Yaskawa INFORM job: long_pipe_cylinder_program.JBI

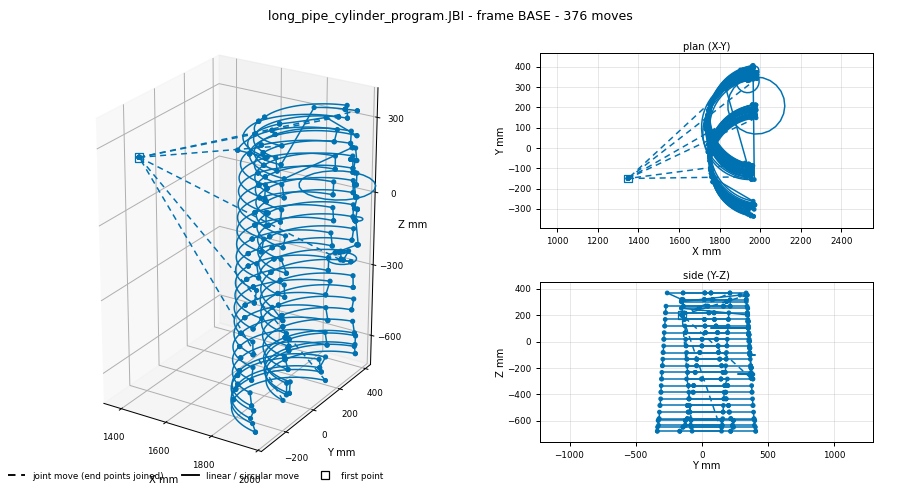
[picture p0: tool path of long_pipe_cylinder_program.JBI in frame BASE, 376 of 498 moves have a stored position in this frame; points joined in program order, loops and branches not executed]
/JOB
//NAME long_pipe_cylinder_program
//POS
///NPOS 488,0,488,1,0,4
///TOOL 0
///POSTYPE BASE
///RECTAN
///RCONF 0,0,0,0,0,0,0,0,0,0,0,0,0,0,0,0,0,0,0,0,0,0,0,0
C00000=1952.474,-141.608,367.212,-93.9778,-89.9999,5.0000
C00001=1952.474,-141.608,367.212,-93.9778,-89.9999,5.0000
C00002=1806.020,-80.138,367.212,-131.5952,-89.9999,5.0000
C00003=1753.400,68.522,367.212,-170.6555,-89.9999,5.0000
C00004=1753.400,68.522,367.212,-170.6555,-89.9999,5.0000
C00005=1753.400,68.522,367.212,-170.6555,-89.9999,5.0000
C00006=1795.925,238.470,367.212,142.2632,-89.9999,5.0000
C00007=1945.817,334.393,367.212,95.8859,-90.0000,5.0000
C00008=1947.913,335.229,317.245,95.3503,-90.0000,5.0000
C00009=1947.913,335.229,317.245,95.3503,-90.0000,5.0000
C00010=1748.482,181.577,317.245,160.6849,-90.0000,5.0000
C00011=1744.683,18.104,317.245,-159.0744,-89.9999,5.0000
C00012=1744.683,18.104,317.245,-159.0744,-89.9999,5.0000
C00013=1744.683,18.104,317.245,-159.0744,-89.9999,5.0000
C00014=1842.190,-106.459,317.245,-121.1710,-89.9999,5.0000
C00015=1928.137,-141.549,317.245,-99.5716,-90.0000,5.0000
C00016=1932.899,-139.870,267.245,-98.5458,-90.0000,5.0000
C00017=1932.899,-139.870,267.245,-98.5458,-90.0000,5.0000
C00018=1770.352,-30.060,267.245,-146.0425,-90.0000,5.0000
C00019=1741.797,163.121,267.245,165.4703,-89.9999,5.0000
C00020=1741.797,163.121,267.245,165.4703,-89.9999,5.0000
C00021=1741.797,163.121,267.245,165.4703,-89.9999,5.0000
C00022=1814.919,283.253,267.245,130.7984,-90.0000,5.0000
C00023=1962.193,340.769,267.245,91.7826,-90.0000,5.0000
C00024=1958.817,343.549,217.245,92.5686,-89.9999,5.0000
C00025=1958.817,343.549,217.245,92.5686,-89.9999,5.0000
C00026=1797.784,264.676,217.245,136.9283,-89.9999,5.0000
C00027=1734.064,92.078,217.245,-177.0797,-89.9999,5.0000
C00028=1734.064,92.078,217.245,-177.0797,-89.9999,5.0000
C00029=1734.064,92.078,217.245,-177.0797,-89.9999,5.0000
C00030=1799.958,-65.427,217.245,-135.0139,-90.0000,5.0000
C00031=1949.378,-134.142,217.245,-94.8421,-90.0000,5.0000
C00032=1957.810,-131.244,167.245,-92.8582,-90.0000,5.0000
C00033=1957.810,-131.244,167.245,-92.8582,-90.0000,5.0000
C00034=1801.335,-64.041,167.245,-135.0154,-89.9999,5.0000
C00035=1735.186,94.868,167.245,-177.7463,-90.0000,5.0000
C00036=1735.186,94.868,167.245,-177.7463,-90.0000,5.0000
C00037=1735.186,94.868,167.245,-177.7463,-90.0000,5.0000
C00038=1799.120,267.709,167.245,136.1700,-90.0000,5.0000
C00039=1966.952,347.413,167.245,90.6138,-90.0000,5.0000
C00040=1967.186,350.732,117.245,90.5513,-90.0000,5.0000
C00041=1967.186,350.732,117.245,90.5513,-90.0000,5.0000
C00042=1802.303,274.899,117.245,134.3981,-89.9999,5.0000
C00043=1734.310,106.876,117.245,179.3219,-89.9999,5.0000
C00044=1734.310,106.876,117.245,179.3219,-89.9999,5.0000
C00045=1734.310,106.876,117.245,179.3219,-89.9999,5.0000
C00046=1803.371,-61.994,117.245,-135.0176,-90.0000,5.0000
C00047=1945.844,-127.883,117.245,-95.8371,-90.0000,5.0000
C00048=1938.801,-124.320,67.245,-97.6695,-90.0000,5.0000
C00049=1938.801,-124.320,67.245,-97.6695,-90.0000,5.0000
C00050=1793.896,-48.619,67.245,-138.9983,-90.0000,5.0000
C00051=1735.617,118.587,67.245,176.4544,-89.9999,5.0000
C00052=1735.617,118.587,67.245,176.4544,-89.9999,5.0000
C00053=1735.617,118.587,67.245,176.4544,-89.9999,5.0000
C00054=1810.878,284.290,67.245,131.3668,-89.9999,5.0000
C00055=1968.204,353.422,67.245,90.3114,-90.0000,5.0000
C00056=1966.949,356.620,17.245,90.5922,-90.0000,5.0000
C00057=1966.949,356.620,17.245,90.5922,-90.0000,5.0000
C00058=1807.041,282.224,17.245,132.3756,-90.0000,5.0000
C00059=1736.566,110.516,17.245,178.4205,-89.9999,5.0000
C00060=1736.566,110.516,17.245,178.4205,-89.9999,5.0000
C00061=1736.566,110.516,17.245,178.4205,-89.9999,5.0000
C00062=1795.050,-47.099,17.245,-139.0948,-90.0000,5.0000
C00063=1959.444,-122.297,17.245,-92.5584,-90.0000,5.0000
C00064=1947.518,-118.948,-32.755,-95.6438,-90.0000,5.0000
C00065=1947.518,-118.948,-32.755,-95.6438,-90.0000,5.0000
C00066=1796.790,-44.821,-32.755,-139.2413,-89.9999,5.0000
C00067=1737.499,122.501,-32.755,175.4642,-90.0000,5.0000
C00068=1737.499,122.501,-32.755,175.4642,-90.0000,5.0000
C00069=1737.499,122.501,-32.755,175.4642,-90.0000,5.0000
C00070=1805.960,284.348,-32.755,132.2266,-89.9999,5.0000
C00071=1967.957,359.139,-32.755,90.3599,-89.9999,5.0000
C00072=1966.253,361.510,-82.755,90.7359,-90.0000,5.0000
C00073=1966.253,361.510,-82.755,90.7359,-90.0000,5.0000
C00074=1815.299,294.981,-82.755,128.9422,-89.9999,5.0000
C00075=1738.257,125.322,-82.755,174.7557,-90.0000,5.0000
C00076=1738.257,125.322,-82.755,174.7557,-90.0000,5.0000
C00077=1738.257,125.322,-82.755,174.7557,-90.0000,5.0000
C00078=1798.652,-42.311,-82.755,-139.4159,-90.0000,5.0000
C00079=1937.806,-115.431,-82.755,-98.2307,-90.0000,5.0000
C00080=1959.669,-113.835,-132.755,-92.5986,-90.0000,5.0000
C00081=1959.669,-113.835,-132.755,-92.5986,-90.0000,5.0000
C00082=1789.517,-29.714,-132.755,-143.3805,-89.9999,5.0000
C00083=1738.347,134.581,-132.755,172.4879,-89.9999,5.0000
C00084=1738.347,134.581,-132.755,172.4879,-89.9999,5.0000
C00085=1738.347,134.581,-132.755,172.4879,-89.9999,5.0000
C00086=1815.608,296.473,-132.755,128.6681,-89.9999,5.0000
C00087=1967.823,365.446,-132.755,90.3807,-90.0000,5.0000
C00088=1960.178,368.374,-182.755,92.0329,-90.0000,5.0000
C00089=1960.178,368.374,-182.755,92.0329,-90.0000,5.0000
C00090=1822.990,305.437,-182.755,126.0528,-90.0000,5.0000
C00091=1740.856,149.131,-182.755,168.8590,-90.0000,5.0000
C00092=1740.856,149.131,-182.755,168.8590,-90.0000,5.0000
C00093=1740.856,149.131,-182.755,168.8590,-90.0000,5.0000
C00094=1790.084,-24.585,-182.755,-144.3607,-90.0000,5.0000
C00095=1949.167,-110.926,-182.755,-95.4178,-90.0000,5.0000
C00096=1949.652,-108.006,-232.755,-95.3619,-89.9999,5.0000
C00097=1949.652,-108.006,-232.755,-95.3619,-89.9999,5.0000
C00098=1790.332,-18.842,-232.755,-145.5533,-89.9999,5.0000
C00099=1742.489,159.932,-232.755,166.1842,-89.9999,5.0000
C00100=1742.489,159.932,-232.755,166.1842,-89.9999,5.0000
C00101=1742.489,159.932,-232.755,166.1842,-89.9999,5.0000
C00102=1820.911,306.183,-232.755,126.3363,-89.9999,5.0000
C00103=1944.457,372.406,-232.755,95.3447,-90.0000,5.0000
C00104=1915.237,385.070,-282.755,100.9422,-90.0000,5.0000
C00105=1915.237,385.070,-282.755,100.9422,-90.0000,5.0000
C00106=1795.330,299.414,-282.755,131.7331,-89.9999,5.0000
C00107=1738.689,144.348,-282.755,170.1088,-89.9999,5.0000
C00108=1738.689,144.348,-282.755,170.1088,-89.9999,5.0000
C00109=1738.689,144.348,-282.755,170.1088,-89.9999,5.0000
C00110=1817.323,-48.028,-282.755,-135.0218,-89.9999,5.0000
C00111=1901.645,-115.476,-282.755,-107.1872,-89.9999,5.0000
C00112=1938.803,-101.562,-332.755,-98.5057,-90.0000,5.0000
C00113=1938.803,-101.562,-332.755,-98.5057,-90.0000,5.0000
C00114=1772.528,11.932,-332.755,-154.9326,-89.9999,5.0000
C00115=1750.419,194.736,-332.755,157.5283,-89.9999,5.0000
C00116=1750.419,194.736,-332.755,157.5283,-89.9999,5.0000
C00117=1750.419,194.736,-332.755,157.5283,-89.9999,5.0000
C00118=1835.466,322.533,-332.755,121.5443,-89.9999,5.0000
C00119=1963.898,376.075,-332.755,91.1925,-90.0000,5.0000
C00120=1964.444,378.545,-382.755,91.0677,-90.0000,5.0000
C00121=1964.444,378.545,-382.755,91.0677,-90.0000,5.0000
C00122=1825.117,315.346,-382.755,124.3619,-90.0000,5.0000
C00123=1748.510,179.382,-382.755,161.1910,-90.0000,5.0000
C00124=1748.510,179.382,-382.755,161.1910,-90.0000,5.0000
C00125=1748.510,179.382,-382.755,161.1910,-90.0000,5.0000
C00126=1783.397,0.464,-382.755,-150.8973,-90.0000,5.0000
C00127=1952.994,-98.481,-382.755,-94.6749,-90.0000,5.0000
C00128=1963.077,-96.189,-432.755,-91.8538,-89.9999,5.0000
C00129=1963.077,-96.189,-432.755,-91.8538,-89.9999,5.0000
C00130=1774.504,19.694,-432.755,-156.6026,-89.9999,5.0000
C00131=1749.909,182.887,-432.755,160.2655,-90.0000,5.0000
C00132=1749.909,182.887,-432.755,160.2655,-90.0000,5.0000
C00133=1749.909,182.887,-432.755,160.2655,-90.0000,5.0000
C00134=1828.820,321.440,-432.755,122.9242,-90.0000,5.0000
C00135=1965.830,382.460,-432.755,90.7675,-89.9999,5.0000
C00136=1956.214,385.900,-482.755,92.7113,-90.0000,5.0000
C00137=1956.214,385.900,-482.755,92.7113,-90.0000,5.0000
C00138=1836.532,331.870,-482.755,120.2857,-89.9999,5.0000
C00139=1754.321,201.072,-482.755,155.7449,-89.9999,5.0000
C00140=1754.321,201.072,-482.755,155.7449,-89.9999,5.0000
C00141=1754.321,201.072,-482.755,155.7449,-89.9999,5.0000
C00142=1775.726,25.199,-482.755,-157.8530,-90.0000,5.0000
C00143=1941.959,-92.060,-482.755,-98.0095,-89.9999,5.0000
C00144=1956.305,-90.288,-532.755,-93.9009,-90.0000,5.0000
C00145=1956.305,-90.288,-532.755,-93.9009,-90.0000,5.0000
C00146=1776.302,28.068,-532.755,-158.5263,-90.0000,5.0000
C00147=1755.401,207.373,-532.755,154.2536,-90.0000,5.0000
C00148=1755.401,207.373,-532.755,154.2536,-90.0000,5.0000
C00149=1755.401,207.373,-532.755,154.2536,-90.0000,5.0000
C00150=1831.521,329.177,-532.755,121.5196,-90.0000,5.0000
C00151=1959.102,390.265,-532.755,92.0928,-89.9999,5.0000
C00152=1966.488,393.604,-582.755,90.6077,-89.9999,5.0000
C00153=1966.488,393.604,-582.755,90.6077,-89.9999,5.0000
C00154=1835.849,336.137,-582.755,119.9516,-90.0000,5.0000
C00155=1758.915,218.913,-582.755,151.4053,-89.9999,5.0000
C00156=1758.915,218.913,-582.755,151.4053,-89.9999,5.0000
C00157=1758.915,218.913,-582.755,151.4053,-89.9999,5.0000
C00158=1768.592,47.728,-582.755,-164.3333,-90.0000,5.0000
C00159=1964.640,-87.533,-582.755,-91.4707,-89.9999,5.0000
C00160=1960.276,-85.309,-632.755,-92.8060,-90.0000,5.0000
C00161=1960.276,-85.309,-632.755,-92.8060,-90.0000,5.0000
C00162=1762.796,68.650,-632.755,-170.2734,-89.9999,5.0000
C00163=1763.792,232.201,-632.755,148.0938,-90.0000,5.0000
C00164=1763.792,232.201,-632.755,148.0938,-90.0000,5.0000
C00165=1763.792,232.201,-632.755,148.0938,-90.0000,5.0000
C00166=1841.674,342.108,-632.755,118.2489,-89.9999,5.0000
C00167=1968.492,396.426,-632.755,90.2093,-90.0000,5.0000
C00168=1968.319,399.205,-596.152,-180.0000,-60.0000,-89.7591
C00169=1968.319,399.205,-596.152,-180.0000,-60.0000,-89.7591
C00170=1843.975,348.228,-596.152,-180.0000,-60.0000,-62.7786
C00171=1766.050,237.566,-596.152,180.0000,-60.0000,-33.2594
C00172=1766.050,237.566,-596.152,180.0000,-60.0000,-33.2594
C00173=1766.050,237.566,-596.152,180.0000,-60.0000,-33.2594
C00174=1763.679,72.740,-596.152,180.0000,-60.0000,8.6585
C00175=1946.255,-81.843,-596.152,180.0000,-60.0000,82.8559
C00176=1943.862,-78.741,-646.152,180.0000,-60.0000,81.9994
C00177=1943.862,-78.741,-646.152,180.0000,-60.0000,81.9994
C00178=1766.299,70.737,-646.152,180.0000,-60.0000,9.3190
C00179=1765.145,237.360,-646.152,180.0000,-60.0000,-33.1025
C00180=1765.145,237.360,-646.152,180.0000,-60.0000,-33.1025
C00181=1765.145,237.360,-646.152,180.0000,-60.0000,-33.1025
C00182=1843.325,349.764,-646.152,180.0000,-60.0000,-62.8045
C00183=1961.291,404.385,-646.152,180.0000,-60.0000,-88.4227
C00184=1965.354,406.519,-677.282,180.0000,-60.0000,-89.2032
C00185=1965.354,406.519,-677.282,180.0000,-60.0000,-89.2032
C00186=1804.746,312.612,-677.282,-180.0000,-60.0000,-51.6774
C00187=1760.400,217.666,-677.282,-180.0000,-60.0000,-28.5021
C00188=1760.400,217.666,-677.282,-180.0000,-60.0000,-28.5021
C00189=1760.400,217.666,-677.282,-180.0000,-60.0000,-28.5021
C00190=1762.623,88.686,-677.282,180.0000,-60.0000,4.2577
C00191=1926.171,-73.826,-677.282,180.0000,-60.0000,76.2948
C00192=1979.466,212.018,367.254,90.2265,-90.0000,5.0000
C00193=1979.466,212.018,367.254,90.2265,-90.0000,5.0000
C00194=1826.445,142.283,367.254,131.1244,-89.9999,5.0000
C00195=1756.890,21.936,367.254,165.9298,-90.0000,5.0000
C00196=1756.890,21.936,367.254,165.9298,-90.0000,5.0000
C00197=1756.890,21.936,367.254,165.9298,-90.0000,5.0000
C00198=1783.627,-126.523,367.254,-154.8432,-90.0000,5.0000
C00199=1965.895,-261.971,367.254,-93.6518,-90.0000,5.0000
C00200=1776.261,-151.339,317.245,-150.1339,-90.0000,5.0000
C00201=1776.261,-151.339,317.245,-150.1339,-90.0000,5.0000
C00202=1753.007,-47.441,317.245,-176.6408,-90.0000,5.0000
C00203=1777.300,81.506,317.245,150.3575,-90.0000,5.0000
C00204=1777.300,81.506,317.245,150.3575,-90.0000,5.0000
C00205=1777.300,81.506,317.245,150.3575,-90.0000,5.0000
C00206=1867.464,176.749,317.245,118.1837,-90.0000,5.0000
C00207=1974.505,213.480,317.245,91.3732,-90.0000,5.0000
C00208=1962.350,213.970,267.245,94.1707,-90.0000,5.0000
C00209=1962.350,213.970,267.245,94.1707,-90.0000,5.0000
C00210=1854.897,163.667,267.245,122.4083,-90.0000,5.0000
C00211=1754.661,45.086,267.245,160.6747,-90.0000,5.0000
C00212=1754.661,45.086,267.245,160.6747,-90.0000,5.0000
C00213=1754.661,45.086,267.245,160.6747,-90.0000,5.0000
C00214=1755.033,-71.682,267.245,-170.5321,-90.0000,5.0000
C00215=1964.286,-271.010,267.245,-93.9005,-89.9999,5.0000
C00216=1964.455,-274.427,217.245,-93.8050,-89.9999,5.0000
C00217=1964.455,-274.427,217.245,-93.8050,-89.9999,5.0000
C00218=1758.542,-91.384,217.245,-165.5228,-89.9999,5.0000
C00219=1766.585,52.944,217.245,157.8540,-90.0000,5.0000
C00220=1766.585,52.944,217.245,157.8540,-90.0000,5.0000
C00221=1766.585,52.944,217.245,157.8540,-90.0000,5.0000
C00222=1856.923,164.760,217.245,121.8464,-90.0000,5.0000
C00223=1973.975,203.799,217.245,91.5566,-90.0000,5.0000
C00224=1976.191,200.287,167.245,91.0384,-90.0000,5.0000
C00225=1976.191,200.287,167.245,91.0384,-90.0000,5.0000
C00226=1844.320,150.002,167.245,126.4793,-90.0000,5.0000
C00227=1756.578,19.544,167.245,166.5261,-89.9999,5.0000
C00228=1756.578,19.544,167.245,166.5261,-89.9999,5.0000
C00229=1756.578,19.544,167.245,166.5261,-89.9999,5.0000
C00230=1763.099,-112.490,167.245,-160.1648,-90.0000,5.0000
C00231=1971.198,-277.055,167.245,-92.1781,-90.0000,5.0000
C00232=1974.265,-280.710,117.245,-91.4340,-90.0000,5.0000
C00233=1974.265,-280.710,117.245,-91.4340,-90.0000,5.0000
C00234=1762.661,-113.911,117.245,-159.8711,-90.0000,5.0000
C00235=1757.863,23.759,117.245,165.4302,-90.0000,5.0000
C00236=1757.863,23.759,117.245,165.4302,-90.0000,5.0000
C00237=1757.863,23.759,117.245,165.4302,-90.0000,5.0000
C00238=1848.435,152.390,117.245,125.2932,-90.0000,5.0000
C00239=1972.348,197.762,117.245,91.9988,-90.0000,5.0000
C00240=1972.379,194.299,67.245,92.0213,-89.9999,5.0000
C00241=1972.379,194.299,67.245,92.0213,-89.9999,5.0000
C00242=1845.484,148.188,67.245,126.5152,-89.9999,5.0000
C00243=1759.522,27.094,67.245,164.5190,-90.0000,5.0000
C00244=1759.522,27.094,67.245,164.5190,-90.0000,5.0000
C00245=1759.522,27.094,67.245,164.5190,-90.0000,5.0000
C00246=1761.533,-113.949,67.245,-159.9578,-90.0000,5.0000
C00247=1967.319,-284.444,67.245,-92.9999,-90.0000,5.0000
C00248=1958.532,-287.141,17.245,-94.9480,-89.9999,5.0000
C00249=1958.532,-287.141,17.245,-94.9480,-89.9999,5.0000
C00250=1764.460,-125.360,17.245,-157.0920,-90.0000,5.0000
C00251=1755.071,1.356,17.245,171.0611,-90.0000,5.0000
C00252=1755.071,1.356,17.245,171.0611,-90.0000,5.0000
C00253=1755.071,1.356,17.245,171.0611,-90.0000,5.0000
C00254=1840.989,140.263,17.245,128.6529,-90.0000,5.0000
C00255=1974.070,191.705,17.245,91.6159,-90.0000,5.0000
C00256=1979.889,188.850,-32.755,90.1413,-90.0000,5.0000
C00257=1979.889,188.850,-32.755,90.1413,-90.0000,5.0000
C00258=1838.594,137.153,-32.755,129.6354,-90.0000,5.0000
C00259=1754.947,0.222,-32.755,171.3474,-89.9999,5.0000
C00260=1754.947,0.222,-32.755,171.3474,-89.9999,5.0000
C00261=1754.947,0.222,-32.755,171.3474,-89.9999,5.0000
C00262=1767.626,-136.866,-32.755,-154.2226,-89.9999,5.0000
C00263=1940.600,-288.358,-32.755,-98.9048,-90.0000,5.0000
C00264=1952.024,-292.820,-82.755,-96.2676,-90.0000,5.0000
C00265=1952.024,-292.820,-82.755,-96.2676,-90.0000,5.0000
C00266=1770.044,-145.488,-82.755,-152.1004,-89.9999,5.0000
C00267=1753.710,-15.340,-82.755,175.2722,-90.0000,5.0000
C00268=1753.710,-15.340,-82.755,175.2722,-90.0000,5.0000
C00269=1753.710,-15.340,-82.755,175.2722,-90.0000,5.0000
C00270=1835.825,132.103,-82.755,131.0279,-89.9999,5.0000
C00271=1971.147,185.827,-82.755,92.4195,-90.0000,5.0000
C00272=1978.997,183.914,-132.755,90.3791,-89.9999,5.0000
C00273=1978.997,183.914,-132.755,90.3791,-89.9999,5.0000
C00274=1817.579,112.933,-132.755,137.9251,-90.0000,5.0000
C00275=1751.687,-39.236,-132.755,-178.7116,-90.0000,5.0000
C00276=1751.687,-39.236,-132.755,-178.7116,-90.0000,5.0000
C00277=1751.687,-39.236,-132.755,-178.7116,-90.0000,5.0000
C00278=1779.686,-169.893,-132.755,-145.9231,-89.9999,5.0000
C00279=1944.840,-295.255,-132.755,-97.7621,-90.0000,5.0000
C00280=1937.661,-298.144,-182.755,-99.2023,-89.9999,5.0000
C00281=1937.661,-298.144,-182.755,-99.2023,-89.9999,5.0000
C00282=1779.767,-171.129,-182.755,-145.6711,-90.0000,5.0000
C00283=1752.198,-39.899,-182.755,-178.5424,-89.9999,5.0000
C00284=1752.198,-39.899,-182.755,-178.5424,-89.9999,5.0000
C00285=1752.198,-39.899,-182.755,-178.5424,-89.9999,5.0000
C00286=1830.409,120.918,-182.755,134.0647,-89.9999,5.0000
C00287=1967.072,180.463,-182.755,93.5650,-90.0000,5.0000
C00288=1967.737,176.940,-232.755,93.4446,-90.0000,5.0000
C00289=1967.737,176.940,-232.755,93.4446,-90.0000,5.0000
C00290=1823.094,112.197,-232.755,137.0853,-90.0000,5.0000
C00291=1752.035,-50.508,-232.755,-175.8889,-90.0000,5.0000
C00292=1752.035,-50.508,-232.755,-175.8889,-90.0000,5.0000
C00293=1752.035,-50.508,-232.755,-175.8889,-90.0000,5.0000
C00294=1786.614,-186.491,-232.755,-141.8229,-90.0000,5.0000
C00295=1970.732,-302.197,-232.755,-92.0736,-90.0000,5.0000
C00296=1936.547,-304.279,-282.755,-99.2272,-90.0000,5.0000
C00297=1936.547,-304.279,-282.755,-99.2272,-90.0000,5.0000
C00298=1775.954,-173.402,-282.755,-145.7345,-89.9999,5.0000
C00299=1751.159,-1.875,-282.755,172.0017,-90.0000,5.0000
C00300=1751.159,-1.875,-282.755,172.0017,-90.0000,5.0000
C00301=1751.159,-1.875,-282.755,172.0017,-90.0000,5.0000
C00302=1855.361,139.589,-282.755,125.7600,-90.0000,5.0000
C00303=1967.526,192.531,-282.755,93.2612,-90.0000,5.0000
C00304=1961.312,172.217,-332.755,95.2969,-89.9999,5.0000
C00305=1961.312,172.217,-332.755,95.2969,-89.9999,5.0000
C00306=1821.236,102.099,-332.755,139.4545,-90.0000,5.0000
C00307=1752.927,-62.146,-332.755,-172.9704,-90.0000,5.0000
C00308=1752.927,-62.146,-332.755,-172.9704,-90.0000,5.0000
C00309=1752.927,-62.146,-332.755,-172.9704,-90.0000,5.0000
C00310=1777.993,-175.868,-332.755,-144.9959,-90.0000,5.0000
C00311=1937.379,-307.215,-332.755,-98.9593,-90.0000,5.0000
C00312=1939.452,-309.026,-382.755,-98.4793,-90.0000,5.0000
C00313=1939.452,-309.026,-382.755,-98.4793,-90.0000,5.0000
C00314=1784.369,-189.678,-382.755,-141.5672,-90.0000,5.0000
C00315=1753.631,-65.654,-382.755,-172.0775,-90.0000,5.0000
C00316=1753.631,-65.654,-382.755,-172.0775,-90.0000,5.0000
C00317=1753.631,-65.654,-382.755,-172.0775,-90.0000,5.0000
C00318=1811.294,87.676,-382.755,144.2498,-90.0000,5.0000
C00319=1965.450,167.920,-382.755,94.2437,-90.0000,5.0000
C00320=1976.104,166.238,-432.755,91.2397,-90.0000,5.0000
C00321=1976.104,166.238,-432.755,91.2397,-90.0000,5.0000
C00322=1797.231,66.653,-432.755,151.1938,-89.9999,5.0000
C00323=1756.658,-97.838,-432.755,-164.0999,-89.9999,5.0000
C00324=1756.658,-97.838,-432.755,-164.0999,-89.9999,5.0000
C00325=1756.658,-97.838,-432.755,-164.0999,-89.9999,5.0000
C00326=1797.206,-217.403,-432.755,-134.9877,-89.9999,5.0000
C00327=1940.733,-311.192,-432.755,-98.1546,-89.9999,5.0000
C00328=1938.247,-316.397,-482.755,-98.5002,-89.9999,5.0000
C00329=1938.247,-316.397,-482.755,-98.5002,-89.9999,5.0000
C00330=1796.071,-218.556,-482.755,-134.9850,-89.9999,5.0000
C00331=1757.920,-109.111,-482.755,-161.3691,-90.0000,5.0000
C00332=1757.920,-109.111,-482.755,-161.3691,-90.0000,5.0000
C00333=1757.920,-109.111,-482.755,-161.3691,-90.0000,5.0000
C00334=1792.221,53.920,-482.755,154.9389,-90.0000,5.0000
C00335=1967.210,162.535,-482.755,93.8491,-90.0000,5.0000
C00336=1978.121,160.335,-532.755,90.6833,-90.0000,5.0000
C00337=1978.121,160.335,-532.755,90.6833,-90.0000,5.0000
C00338=1794.434,54.529,-532.755,154.5248,-89.9999,5.0000
C00339=1758.419,-102.880,-532.755,-162.7854,-90.0000,5.0000
C00340=1758.419,-102.880,-532.755,-162.7854,-90.0000,5.0000
C00341=1758.419,-102.880,-532.755,-162.7854,-90.0000,5.0000
C00342=1790.443,-210.664,-532.755,-137.0973,-90.0000,5.0000
C00343=1934.317,-320.451,-532.755,-99.1497,-89.9999,5.0000
C00344=1942.640,-323.151,-582.755,-97.4501,-90.0000,5.0000
C00345=1942.640,-323.151,-582.755,-97.4501,-90.0000,5.0000
C00346=1801.232,-230.128,-582.755,-132.4320,-89.9999,5.0000
C00347=1757.450,-110.352,-582.755,-161.1196,-90.0000,5.0000
C00348=1757.450,-110.352,-582.755,-161.1196,-90.0000,5.0000
C00349=1757.450,-110.352,-582.755,-161.1196,-90.0000,5.0000
C00350=1788.731,43.478,-582.755,157.9704,-89.9999,5.0000
C00351=1973.897,157.381,-582.755,91.9568,-89.9999,5.0000
C00352=1951.154,153.676,-632.755,98.8647,-90.0000,5.0000
C00353=1951.154,153.676,-632.755,98.8647,-90.0000,5.0000
C00354=1786.262,35.054,-632.755,160.3992,-90.0000,5.0000
C00355=1760.007,-125.303,-632.755,-157.5209,-90.0000,5.0000
C00356=1760.007,-125.303,-632.755,-157.5209,-90.0000,5.0000
C00357=1760.007,-125.303,-632.755,-157.5209,-90.0000,5.0000
C00358=1800.669,-233.671,-632.755,-132.0108,-90.0000,5.0000
C00359=1940.775,-327.209,-632.755,-97.7064,-90.0000,5.0000
C00360=1955.591,-329.848,-596.152,180.0000,-60.0000,85.1975
C00361=1955.591,-329.848,-596.152,180.0000,-60.0000,85.1975
C00362=1799.504,-233.466,-596.152,-180.0000,-60.0000,47.7757
C00363=1759.022,-124.965,-596.152,180.0000,-60.0000,22.3141
C00364=1759.022,-124.965,-596.152,180.0000,-60.0000,22.3141
C00365=1759.022,-124.965,-596.152,180.0000,-60.0000,22.3141
C00366=1783.812,27.666,-596.152,180.0000,-60.0000,-17.4368
C00367=1949.732,150.709,-596.152,-180.0000,-60.0000,-80.5655
C00368=1960.973,149.730,-646.152,180.0000,-60.0000,-83.9551
C00369=1960.973,149.730,-646.152,180.0000,-60.0000,-83.9551
C00370=1776.817,10.663,-646.152,-180.0000,-60.0000,-12.3962
C00371=1761.547,-142.155,-646.152,-180.0000,-60.0000,26.2748
C00372=1761.547,-142.155,-646.152,-180.0000,-60.0000,26.2748
C00373=1761.547,-142.155,-646.152,-180.0000,-60.0000,26.2748
C00374=1806.157,-244.506,-646.152,180.0000,-60.0000,50.3655
C00375=1954.328,-334.905,-646.152,-180.0000,-60.0000,85.0389
C00376=1967.761,-336.723,-677.101,180.0000,-60.0000,87.6009
C00377=1967.761,-336.723,-677.101,180.0000,-60.0000,87.6009
C00378=1815.884,-252.718,-677.101,180.0000,-60.0000,53.0321
C00379=1767.098,-166.865,-677.101,-180.0000,-60.0000,31.8961
C00380=1767.098,-166.865,-677.101,-180.0000,-60.0000,31.8961
C00381=1767.098,-166.865,-677.101,-180.0000,-60.0000,31.8961
C00382=1769.939,-14.132,-677.101,180.0000,-60.0000,-5.4166
C00383=1980.328,148.699,-677.101,180.0000,-60.0000,-89.9650
C00384=1984.725,342.559,351.030,90.0895,-90.0000,5.0000
C00385=1984.725,342.559,351.030,90.0895,-90.0000,5.0000
C00386=1951.125,337.003,351.030,98.9805,-89.9999,5.0000
C00387=1938.621,333.209,351.030,102.4149,-89.9999,5.0000
C00388=1938.621,333.209,351.030,102.4149,-89.9999,5.0000
C00389=1938.621,333.209,351.030,102.4149,-89.9999,5.0000
C00390=1882.277,317.051,351.030,117.8151,-90.0000,5.0000
C00391=1832.895,288.262,351.030,132.5031,-90.0000,5.0000
C00392=1958.049,-155.412,301.930,-95.5589,-90.0000,5.0000
C00393=1958.049,-155.412,301.930,-95.5589,-90.0000,5.0000
C00394=1730.330,0.812,301.930,-154.5192,-90.0000,5.0000
C00395=1746.203,186.558,301.930,164.9234,-90.0000,5.0000
C00396=1746.203,186.558,301.930,164.9234,-90.0000,5.0000
C00397=1746.203,186.558,301.930,164.9234,-90.0000,5.0000
C00398=1835.265,302.972,301.930,129.6502,-89.9999,5.0000
C00399=1857.274,335.764,301.930,120.8974,-90.0000,5.0000
C00400=1982.982,346.261,251.930,90.5338,-90.0000,5.0000
C00401=1982.982,346.261,251.930,90.5338,-90.0000,5.0000
C00402=1711.972,113.746,251.930,-178.2245,-90.0000,5.0000
C00403=1743.833,-19.410,251.930,-149.5841,-90.0000,5.0000
C00404=1743.833,-19.410,251.930,-149.5841,-90.0000,5.0000
C00405=1743.833,-19.410,251.930,-149.5841,-90.0000,5.0000
C00406=1839.889,-116.346,251.930,-121.3236,-90.0000,5.0000
C00407=1971.426,-155.384,251.930,-92.8137,-90.0000,5.0000
C00408=1965.864,344.090,201.930,94.9470,-90.0000,5.0000
C00409=1965.864,344.090,201.930,94.9470,-90.0000,5.0000
C00410=1967.949,344.857,201.930,94.3970,-90.0000,5.0000
C00411=1967.674,345.019,201.930,94.4643,-90.0000,5.0000
C00412=1967.674,345.019,201.930,94.4643,-90.0000,5.0000
C00413=1967.674,345.019,201.930,94.4643,-90.0000,5.0000
C00414=1969.158,345.300,201.930,94.0795,-90.0000,5.0000
C00415=1978.854,346.488,201.930,91.5874,-90.0000,5.0000
C00416=1982.729,350.115,151.930,90.5883,-90.0000,5.0000
C00417=1982.729,350.115,151.930,90.5883,-90.0000,5.0000
C00418=1971.147,349.465,151.930,93.5057,-90.0000,5.0000
C00419=1958.305,348.424,151.930,96.7476,-90.0000,5.0000
C00420=1958.305,348.424,151.930,96.7476,-90.0000,5.0000
C00421=1958.305,348.424,151.930,96.7476,-90.0000,5.0000
C00422=1966.090,347.909,151.930,94.8068,-90.0000,5.0000
C00423=1977.443,347.873,151.930,91.9356,-89.9999,5.0000
C00424=1968.045,349.288,101.930,94.2875,-89.9999,5.0000
C00425=1968.045,349.288,101.930,94.2875,-89.9999,5.0000
C00426=1983.428,349.890,101.930,90.4130,-90.0000,5.0000
C00427=1976.137,349.815,101.930,92.2473,-90.0000,5.0000
C00428=1976.137,349.815,101.930,92.2473,-90.0000,5.0000
C00429=1976.137,349.815,101.930,92.2473,-90.0000,5.0000
C00430=1982.494,350.032,101.930,90.6477,-89.9999,5.0000
C00431=1984.894,350.113,101.930,90.0441,-90.0000,5.0000
C00432=1980.139,356.174,51.930,91.2071,-90.0000,5.0000
C00433=1980.139,356.174,51.930,91.2071,-90.0000,5.0000
C00434=1975.906,355.661,51.930,92.2477,-90.0000,5.0000
C00435=1973.661,354.809,51.930,92.8079,-90.0000,5.0000
C00436=1973.661,354.809,51.930,92.8079,-90.0000,5.0000
C00437=1973.661,354.809,51.930,92.8079,-90.0000,5.0000
C00438=1967.304,354.361,51.930,94.3760,-90.0000,5.0000
C00439=1973.731,353.378,51.930,92.8080,-90.0000,5.0000
C00440=1978.040,356.452,1.930,91.7188,-90.0000,5.0000
C00441=1978.040,356.452,1.930,91.7188,-90.0000,5.0000
C00442=1979.225,356.894,1.930,91.4265,-90.0000,5.0000
C00443=1977.244,357.995,1.930,91.9010,-90.0000,5.0000
C00444=1977.244,357.995,1.930,91.9010,-90.0000,5.0000
C00445=1977.244,357.995,1.930,91.9010,-90.0000,5.0000
C00446=1982.820,358.225,1.930,90.5461,-90.0000,5.0000
C00447=1983.072,358.586,1.930,90.4841,-90.0000,5.0000
C00448=1971.386,362.062,-48.070,93.2652,-89.9999,5.0000
C00449=1971.386,362.062,-48.070,93.2652,-89.9999,5.0000
C00450=1984.157,361.226,-48.070,90.2188,-89.9999,5.0000
C00451=1984.157,361.226,-48.070,90.2188,-89.9999,5.0000
C00452=1984.157,361.226,-48.070,90.2188,-89.9999,5.0000
C00453=1984.157,361.226,-48.070,90.2188,-89.9999,5.0000
C00454=1984.157,361.226,-48.070,90.2188,-89.9999,5.0000
C00455=1984.157,361.226,-48.070,90.2188,-89.9999,5.0000
C00456=1974.928,363.021,-98.070,92.4115,-90.0000,5.0000
C00457=1974.928,363.021,-98.070,92.4115,-90.0000,5.0000
C00458=1965.376,362.677,-98.070,94.6820,-90.0000,5.0000
C00459=1975.510,363.443,-98.070,92.2693,-89.9999,5.0000
C00460=1975.510,363.443,-98.070,92.2693,-89.9999,5.0000
C00461=1975.510,363.443,-98.070,92.2693,-89.9999,5.0000
C00462=1972.062,363.413,-98.070,93.0868,-90.0000,5.0000
C00463=1977.715,363.777,-98.070,91.7439,-90.0000,5.0000
C00464=1984.970,373.050,-198.070,90.0227,-90.0000,5.0000
C00465=1984.970,373.050,-198.070,90.0227,-90.0000,5.0000
C00466=1981.006,371.625,-198.070,90.9334,-90.0000,5.0000
C00467=1981.006,371.625,-198.070,90.9334,-90.0000,5.0000
C00468=1981.006,371.625,-198.070,90.9334,-90.0000,5.0000
C00469=1981.006,371.625,-198.070,90.9334,-90.0000,5.0000
C00470=1981.006,371.625,-198.070,90.9334,-90.0000,5.0000
C00471=1981.006,371.625,-198.070,90.9334,-90.0000,5.0000
C00472=1892.586,361.867,-248.070,111.1017,-90.0000,5.0000
C00473=1892.586,361.867,-248.070,111.1017,-90.0000,5.0000
C00474=1969.935,376.419,-248.070,93.4071,-90.0000,5.0000
C00475=1903.290,373.261,-248.070,108.0431,-90.0000,5.0000
C00476=1903.290,373.261,-248.070,108.0431,-90.0000,5.0000
C00477=1903.290,373.261,-248.070,108.0431,-90.0000,5.0000
C00478=1925.960,378.588,-248.070,102.9831,-90.0000,5.0000
C00479=1903.410,384.950,-248.070,107.2653,-90.0000,5.0000
C00480=1909.717,376.985,-277.282,106.4763,-90.0000,5.0000
C00481=1909.717,376.985,-277.282,106.4763,-90.0000,5.0000
C00482=1919.584,375.149,-277.282,104.5151,-90.0000,5.0000
C00483=1952.993,376.996,-277.282,97.1756,-90.0000,5.0000
C00484=1952.993,376.996,-277.282,97.1756,-90.0000,5.0000
C00485=1952.993,376.996,-277.282,97.1756,-90.0000,5.0000
C00486=1932.130,374.374,-277.282,101.8565,-89.9999,5.0000
C00487=1911.505,370.674,-277.282,106.4929,-90.0000,5.0000
///POSTYPE PULSE
///PULSE
EC00000=0
EC00001=0
EC00002=0
EC00003=0
EC00004=0
EC00005=0
EC00006=0
EC00007=0
EC00008=0
EC00009=0
EC00010=0
EC00011=0
EC00012=0
EC00013=0
EC00014=0
EC00015=0
EC00016=0
EC00017=0
EC00018=0
EC00019=0
EC00020=0
EC00021=0
EC00022=0
EC00023=0
EC00024=0
EC00025=0
EC00026=0
EC00027=0
EC00028=0
EC00029=0
EC00030=0
EC00031=0
EC00032=0
EC00033=0
EC00034=0
EC00035=0
EC00036=0
EC00037=0
EC00038=0
EC00039=0
EC00040=0
EC00041=0
EC00042=0
EC00043=0
EC00044=0
EC00045=0
EC00046=0
EC00047=0
EC00048=0
EC00049=0
EC00050=0
EC00051=0
EC00052=0
EC00053=0
EC00054=0
EC00055=0
EC00056=0
EC00057=0
EC00058=0
EC00059=0
EC00060=0
EC00061=0
EC00062=0
EC00063=0
EC00064=0
EC00065=0
EC00066=0
EC00067=0
EC00068=0
EC00069=0
EC00070=0
EC00071=0
EC00072=0
EC00073=0
EC00074=0
EC00075=0
EC00076=0
EC00077=0
EC00078=0
EC00079=0
EC00080=0
EC00081=0
EC00082=0
EC00083=0
EC00084=0
EC00085=0
EC00086=0
EC00087=0
EC00088=0
EC00089=0
EC00090=0
EC00091=0
EC00092=0
EC00093=0
EC00094=0
EC00095=0
EC00096=0
EC00097=0
EC00098=0
EC00099=0
EC00100=0
EC00101=0
EC00102=0
EC00103=0
EC00104=0
EC00105=0
EC00106=0
EC00107=0
EC00108=0
EC00109=0
EC00110=0
EC00111=0
EC00112=0
EC00113=0
EC00114=0
EC00115=0
EC00116=0
EC00117=0
EC00118=0
EC00119=0
EC00120=0
EC00121=0
EC00122=0
EC00123=0
EC00124=0
EC00125=0
EC00126=0
EC00127=0
EC00128=0
EC00129=0
EC00130=0
EC00131=0
EC00132=0
EC00133=0
EC00134=0
EC00135=0
EC00136=0
EC00137=0
EC00138=0
EC00139=0
EC00140=0
EC00141=0
EC00142=0
EC00143=0
EC00144=0
EC00145=0
EC00146=0
EC00147=0
EC00148=0
EC00149=0
EC00150=0
EC00151=0
EC00152=0
EC00153=0
EC00154=0
EC00155=0
EC00156=0
EC00157=0
EC00158=0
EC00159=0
EC00160=0
EC00161=0
EC00162=0
EC00163=0
EC00164=0
EC00165=0
EC00166=0
EC00167=0
EC00168=0
EC00169=0
EC00170=0
EC00171=0
EC00172=0
EC00173=0
EC00174=0
EC00175=0
EC00176=0
EC00177=0
EC00178=0
EC00179=0
EC00180=0
EC00181=0
EC00182=0
EC00183=0
EC00184=0
EC00185=0
EC00186=0
EC00187=0
EC00188=0
EC00189=0
EC00190=0
EC00191=0
EC00192=184320
EC00193=184320
EC00194=184320
EC00195=184320
EC00196=184320
EC00197=184320
EC00198=184320
EC00199=184320
EC00200=184320
EC00201=184320
EC00202=184320
EC00203=184320
EC00204=184320
EC00205=184320
EC00206=184320
EC00207=184320
EC00208=184320
EC00209=184320
EC00210=184320
EC00211=184320
EC00212=184320
EC00213=184320
EC00214=184320
EC00215=184320
EC00216=184320
EC00217=184320
EC00218=184320
EC00219=184320
EC00220=184320
EC00221=184320
EC00222=184320
EC00223=184320
EC00224=184320
EC00225=184320
EC00226=184320
EC00227=184320
EC00228=184320
EC00229=184320
EC00230=184320
EC00231=184320
EC00232=184320
EC00233=184320
EC00234=184320
EC00235=184320
EC00236=184320
EC00237=184320
EC00238=184320
EC00239=184320
EC00240=184320
EC00241=184320
EC00242=184320
EC00243=184320
EC00244=184320
EC00245=184320
EC00246=184320
EC00247=184320
EC00248=184320
EC00249=184320
EC00250=184320
EC00251=184320
EC00252=184320
EC00253=184320
EC00254=184320
EC00255=184320
EC00256=184320
EC00257=184320
EC00258=184320
EC00259=184320
EC00260=184320
EC00261=184320
EC00262=184320
EC00263=184320
EC00264=184320
EC00265=184320
EC00266=184320
EC00267=184320
EC00268=184320
EC00269=184320
EC00270=184320
EC00271=184320
EC00272=184320
EC00273=184320
EC00274=184320
EC00275=184320
EC00276=184320
EC00277=184320
EC00278=184320
EC00279=184320
EC00280=184320
EC00281=184320
EC00282=184320
EC00283=184320
EC00284=184320
EC00285=184320
EC00286=184320
EC00287=184320
EC00288=184320
EC00289=184320
EC00290=184320
EC00291=184320
EC00292=184320
EC00293=184320
EC00294=184320
EC00295=184320
EC00296=184320
EC00297=184320
EC00298=184320
EC00299=184320
EC00300=184320
EC00301=184320
EC00302=184320
EC00303=184320
EC00304=184320
EC00305=184320
EC00306=184320
EC00307=184320
EC00308=184320
EC00309=184320
EC00310=184320
EC00311=184320
EC00312=184320
EC00313=184320
EC00314=184320
EC00315=184320
EC00316=184320
EC00317=184320
EC00318=184320
EC00319=184320
EC00320=184320
EC00321=184320
EC00322=184320
EC00323=184320
EC00324=184320
EC00325=184320
EC00326=184320
EC00327=184320
EC00328=184320
EC00329=184320
EC00330=184320
EC00331=184320
EC00332=184320
EC00333=184320
EC00334=184320
EC00335=184320
EC00336=184320
EC00337=184320
EC00338=184320
EC00339=184320
EC00340=184320
EC00341=184320
EC00342=184320
EC00343=184320
EC00344=184320
EC00345=184320
EC00346=184320
EC00347=184320
EC00348=184320
EC00349=184320
EC00350=184320
EC00351=184320
EC00352=184320
EC00353=184320
EC00354=184320
EC00355=184320
EC00356=184320
EC00357=184320
EC00358=184320
EC00359=184320
EC00360=184320
EC00361=184320
EC00362=184320
EC00363=184320
EC00364=184320
EC00365=184320
EC00366=184320
EC00367=184320
EC00368=184320
EC00369=184320
EC00370=184320
EC00371=184320
EC00372=184320
EC00373=184320
EC00374=184320
EC00375=184320
EC00376=184320
EC00377=184320
EC00378=184320
EC00379=184320
EC00380=184320
EC00381=184320
EC00382=184320
EC00383=184320
EC00384=276480
EC00385=276480
EC00386=276480
EC00387=276480
EC00388=276480
EC00389=276480
EC00390=276480
EC00391=276480
EC00392=276480
EC00393=276480
EC00394=276480
EC00395=276480
EC00396=276480
EC00397=276480
EC00398=276480
EC00399=276480
EC00400=276480
EC00401=276480
EC00402=276480
EC00403=276480
EC00404=276480
EC00405=276480
EC00406=276480
EC00407=276480
EC00408=276480
EC00409=276480
EC00410=276480
EC00411=276480
EC00412=276480
EC00413=276480
EC00414=276480
EC00415=276480
EC00416=276480
EC00417=276480
EC00418=276480
EC00419=276480
EC00420=276480
EC00421=276480
EC00422=276480
EC00423=276480
EC00424=276480
EC00425=276480
EC00426=276480
EC00427=276480
EC00428=276480
EC00429=276480
EC00430=276480
EC00431=276480
EC00432=276480
EC00433=276480
EC00434=276480
EC00435=276480
EC00436=276480
EC00437=276480
EC00438=276480
EC00439=276480
EC00440=276480
EC00441=276480
EC00442=276480
EC00443=276480
EC00444=276480
EC00445=276480
EC00446=276480
EC00447=276480
EC00448=276480
EC00449=276480
EC00450=276480
EC00451=276480
EC00452=276480
EC00453=276480
EC00454=276480
EC00455=276480
EC00456=276480
EC00457=276480
EC00458=276480
EC00459=276480
EC00460=276480
EC00461=276480
EC00462=276480
EC00463=276480
EC00464=276480
EC00465=276480
EC00466=276480
EC00467=276480
EC00468=276480
EC00469=276480
EC00470=276480
EC00471=276480
EC00472=276480
EC00473=276480
EC00474=276480
EC00475=276480
EC00476=276480
EC00477=276480
EC00478=276480
EC00479=276480
EC00480=276480
EC00481=276480
EC00482=276480
EC00483=276480
EC00484=276480
EC00485=276480
EC00486=276480
EC00487=276480
///POSTYPE BASE
///RECTAN
///RCONF 1,0,0,0,0,0,0,0,0,0,0,0,0,0,0,0,0,0,0,0,0,0,0,0
P00009=1350.000,-150.000,200.000,-180.0000,-45.0000,0.0000
///POSTYPE PULSE
///PULSE
EX00000=92160
EX00001=184320
EX00002=276480
EX00003=368640
//INST
///DATE 2023/07/11 13:37
///ATTR SC,RW,RJ
////FRAME BASE
///GROUP1 RB1,ST1
NOP
MOVJ P009 EX000 VJ=15.00
MOVJ P009 VJ=15.00
MOVJ C00000 EC00000 VJ=15.00
CALL JOB:SPYON
MOVC C00001 EC00001 V=150.0
MOVC C00002 EC00002 V=150.0
MOVC C00003 EC00003 V=150.0
MOVL C00004 EC00004 V=150.0
MOVC C00005 EC00005 V=150.0
MOVC C00006 EC00006 V=150.0
MOVC C00007 EC00007 V=150.0
MOVL C00008 EC00008 V=150.0
MOVC C00009 EC00009 V=150.0
MOVC C00010 EC00010 V=150.0
MOVC C00011 EC00011 V=150.0
MOVL C00012 EC00012 V=150.0
MOVC C00013 EC00013 V=150.0
MOVC C00014 EC00014 V=150.0
MOVC C00015 EC00015 V=150.0
MOVL C00016 EC00016 V=150.0
MOVC C00017 EC00017 V=150.0
MOVC C00018 EC00018 V=150.0
MOVC C00019 EC00019 V=150.0
MOVL C00020 EC00020 V=150.0
MOVC C00021 EC00021 V=150.0
MOVC C00022 EC00022 V=150.0
MOVC C00023 EC00023 V=150.0
MOVL C00024 EC00024 V=150.0
MOVC C00025 EC00025 V=150.0
MOVC C00026 EC00026 V=150.0
MOVC C00027 EC00027 V=150.0
MOVL C00028 EC00028 V=150.0
MOVC C00029 EC00029 V=150.0
MOVC C00030 EC00030 V=150.0
MOVC C00031 EC00031 V=150.0
MOVL C00032 EC00032 V=150.0
MOVC C00033 EC00033 V=150.0
MOVC C00034 EC00034 V=150.0
MOVC C00035 EC00035 V=150.0
MOVL C00036 EC00036 V=150.0
MOVC C00037 EC00037 V=150.0
MOVC C00038 EC00038 V=150.0
MOVC C00039 EC00039 V=150.0
MOVL C00040 EC00040 V=150.0
MOVC C00041 EC00041 V=150.0
MOVC C00042 EC00042 V=150.0
MOVC C00043 EC00043 V=150.0
MOVL C00044 EC00044 V=150.0
MOVC C00045 EC00045 V=150.0
MOVC C00046 EC00046 V=150.0
MOVC C00047 EC00047 V=150.0
MOVL C00048 EC00048 V=150.0
MOVC C00049 EC00049 V=150.0
MOVC C00050 EC00050 V=150.0
MOVC C00051 EC00051 V=150.0
MOVL C00052 EC00052 V=150.0
MOVC C00053 EC00053 V=150.0
MOVC C00054 EC00054 V=150.0
MOVC C00055 EC00055 V=150.0
MOVL C00056 EC00056 V=150.0
MOVC C00057 EC00057 V=150.0
MOVC C00058 EC00058 V=150.0
MOVC C00059 EC00059 V=150.0
MOVL C00060 EC00060 V=150.0
MOVC C00061 EC00061 V=150.0
MOVC C00062 EC00062 V=150.0
MOVC C00063 EC00063 V=150.0
MOVL C00064 EC00064 V=150.0
MOVC C00065 EC00065 V=150.0
MOVC C00066 EC00066 V=150.0
MOVC C00067 EC00067 V=150.0
MOVL C00068 EC00068 V=150.0
MOVC C00069 EC00069 V=150.0
MOVC C00070 EC00070 V=150.0
MOVC C00071 EC00071 V=150.0
MOVL C00072 EC00072 V=150.0
MOVC C00073 EC00073 V=150.0
MOVC C00074 EC00074 V=150.0
MOVC C00075 EC00075 V=150.0
MOVL C00076 EC00076 V=150.0
MOVC C00077 EC00077 V=150.0
MOVC C00078 EC00078 V=150.0
MOVC C00079 EC00079 V=150.0
MOVL C00080 EC00080 V=150.0
MOVC C00081 EC00081 V=150.0
MOVC C00082 EC00082 V=150.0
MOVC C00083 EC00083 V=150.0
MOVL C00084 EC00084 V=150.0
MOVC C00085 EC00085 V=150.0
MOVC C00086 EC00086 V=150.0
MOVC C00087 EC00087 V=150.0
MOVL C00088 EC00088 V=150.0
MOVC C00089 EC00089 V=150.0
MOVC C00090 EC00090 V=150.0
MOVC C00091 EC00091 V=150.0
MOVL C00092 EC00092 V=150.0
MOVC C00093 EC00093 V=150.0
MOVC C00094 EC00094 V=150.0
MOVC C00095 EC00095 V=150.0
MOVL C00096 EC00096 V=150.0
MOVC C00097 EC00097 V=150.0
MOVC C00098 EC00098 V=150.0
MOVC C00099 EC00099 V=150.0
MOVL C00100 EC00100 V=150.0
MOVC C00101 EC00101 V=150.0
MOVC C00102 EC00102 V=150.0
MOVC C00103 EC00103 V=150.0
MOVL C00104 EC00104 V=150.0
MOVC C00105 EC00105 V=150.0
MOVC C00106 EC00106 V=150.0
MOVC C00107 EC00107 V=150.0
MOVL C00108 EC00108 V=150.0
MOVC C00109 EC00109 V=150.0
MOVC C00110 EC00110 V=150.0
MOVC C00111 EC00111 V=150.0
MOVL C00112 EC00112 V=150.0
MOVC C00113 EC00113 V=150.0
MOVC C00114 EC00114 V=150.0
MOVC C00115 EC00115 V=150.0
MOVL C00116 EC00116 V=150.0
MOVC C00117 EC00117 V=150.0
MOVC C00118 EC00118 V=150.0
MOVC C00119 EC00119 V=150.0
MOVL C00120 EC00120 V=150.0
MOVC C00121 EC00121 V=150.0
MOVC C00122 EC00122 V=150.0
MOVC C00123 EC00123 V=150.0
MOVL C00124 EC00124 V=150.0
MOVC C00125 EC00125 V=150.0
MOVC C00126 EC00126 V=150.0
MOVC C00127 EC00127 V=150.0
MOVL C00128 EC00128 V=150.0
MOVC C00129 EC00129 V=150.0
MOVC C00130 EC00130 V=150.0
MOVC C00131 EC00131 V=150.0
MOVL C00132 EC00132 V=150.0
MOVC C00133 EC00133 V=150.0
MOVC C00134 EC00134 V=150.0
MOVC C00135 EC00135 V=150.0
MOVL C00136 EC00136 V=150.0
MOVC C00137 EC00137 V=150.0
MOVC C00138 EC00138 V=150.0
MOVC C00139 EC00139 V=150.0
MOVL C00140 EC00140 V=150.0
MOVC C00141 EC00141 V=150.0
MOVC C00142 EC00142 V=150.0
MOVC C00143 EC00143 V=150.0
MOVL C00144 EC00144 V=150.0
MOVC C00145 EC00145 V=150.0
MOVC C00146 EC00146 V=150.0
MOVC C00147 EC00147 V=150.0
MOVL C00148 EC00148 V=150.0
MOVC C00149 EC00149 V=150.0
MOVC C00150 EC00150 V=150.0
MOVC C00151 EC00151 V=150.0
MOVL C00152 EC00152 V=150.0
MOVC C00153 EC00153 V=150.0
MOVC C00154 EC00154 V=150.0
MOVC C00155 EC00155 V=150.0
MOVL C00156 EC00156 V=150.0
MOVC C00157 EC00157 V=150.0
MOVC C00158 EC00158 V=150.0
MOVC C00159 EC00159 V=150.0
MOVL C00160 EC00160 V=150.0
MOVC C00161 EC00161 V=150.0
MOVC C00162 EC00162 V=150.0
MOVC C00163 EC00163 V=150.0
MOVL C00164 EC00164 V=150.0
MOVC C00165 EC00165 V=150.0
MOVC C00166 EC00166 V=150.0
MOVC C00167 EC00167 V=150.0
MOVL C00168 EC00168 V=150.0
MOVC C00169 EC00169 V=150.0
MOVC C00170 EC00170 V=150.0
MOVC C00171 EC00171 V=150.0
MOVL C00172 EC00172 V=150.0
MOVC C00173 EC00173 V=150.0
MOVC C00174 EC00174 V=150.0
MOVC C00175 EC00175 V=150.0
MOVL C00176 EC00176 V=150.0
MOVC C00177 EC00177 V=150.0
MOVC C00178 EC00178 V=150.0
MOVC C00179 EC00179 V=150.0
MOVL C00180 EC00180 V=150.0
MOVC C00181 EC00181 V=150.0
MOVC C00182 EC00182 V=150.0
MOVC C00183 EC00183 V=150.0
MOVL C00184 EC00184 V=150.0
MOVC C00185 EC00185 V=150.0
MOVC C00186 EC00186 V=150.0
MOVC C00187 EC00187 V=150.0
MOVL C00188 EC00188 V=150.0
MOVC C00189 EC00189 V=150.0
MOVC C00190 EC00190 V=150.0
MOVC C00191 EC00191 V=150.0
CALL JOB:SPYOF
MOVJ P009 VJ=15.00
MOVL P009 EX000 V=150.0
MOVJ P009 VJ=15.00
MOVL P009 EX001 V=150.0
MOVJ C00192 EC00192 VJ=15.00
CALL JOB:SPYON
MOVC C00193 EC00193 V=150.0
MOVC C00194 EC00194 V=150.0
MOVC C00195 EC00195 V=150.0
MOVL C00196 EC00196 V=150.0
MOVC C00197 EC00197 V=150.0
MOVC C00198 EC00198 V=150.0
MOVC C00199 EC00199 V=150.0
MOVL C00200 EC00200 V=150.0
MOVC C00201 EC00201 V=150.0
MOVC C00202 EC00202 V=150.0
MOVC C00203 EC00203 V=150.0
MOVL C00204 EC00204 V=150.0
MOVC C00205 EC00205 V=150.0
MOVC C00206 EC00206 V=150.0
MOVC C00207 EC00207 V=150.0
MOVL C00208 EC00208 V=150.0
MOVC C00209 EC00209 V=150.0
MOVC C00210 EC00210 V=150.0
MOVC C00211 EC00211 V=150.0
MOVL C00212 EC00212 V=150.0
MOVC C00213 EC00213 V=150.0
MOVC C00214 EC00214 V=150.0
MOVC C00215 EC00215 V=150.0
MOVL C00216 EC00216 V=150.0
MOVC C00217 EC00217 V=150.0
MOVC C00218 EC00218 V=150.0
MOVC C00219 EC00219 V=150.0
MOVL C00220 EC00220 V=150.0
MOVC C00221 EC00221 V=150.0
MOVC C00222 EC00222 V=150.0
MOVC C00223 EC00223 V=150.0
MOVL C00224 EC00224 V=150.0
MOVC C00225 EC00225 V=150.0
MOVC C00226 EC00226 V=150.0
MOVC C00227 EC00227 V=150.0
MOVL C00228 EC00228 V=150.0
MOVC C00229 EC00229 V=150.0
MOVC C00230 EC00230 V=150.0
MOVC C00231 EC00231 V=150.0
MOVL C00232 EC00232 V=150.0
MOVC C00233 EC00233 V=150.0
MOVC C00234 EC00234 V=150.0
MOVC C00235 EC00235 V=150.0
MOVL C00236 EC00236 V=150.0
MOVC C00237 EC00237 V=150.0
MOVC C00238 EC00238 V=150.0
MOVC C00239 EC00239 V=150.0
MOVL C00240 EC00240 V=150.0
MOVC C00241 EC00241 V=150.0
MOVC C00242 EC00242 V=150.0
MOVC C00243 EC00243 V=150.0
MOVL C00244 EC00244 V=150.0
MOVC C00245 EC00245 V=150.0
MOVC C00246 EC00246 V=150.0
MOVC C00247 EC00247 V=150.0
MOVL C00248 EC00248 V=150.0
MOVC C00249 EC00249 V=150.0
MOVC C00250 EC00250 V=150.0
MOVC C00251 EC00251 V=150.0
MOVL C00252 EC00252 V=150.0
MOVC C00253 EC00253 V=150.0
MOVC C00254 EC00254 V=150.0
MOVC C00255 EC00255 V=150.0
MOVL C00256 EC00256 V=150.0
MOVC C00257 EC00257 V=150.0
MOVC C00258 EC00258 V=150.0
MOVC C00259 EC00259 V=150.0
MOVL C00260 EC00260 V=150.0
MOVC C00261 EC00261 V=150.0
MOVC C00262 EC00262 V=150.0
MOVC C00263 EC00263 V=150.0
MOVL C00264 EC00264 V=150.0
MOVC C00265 EC00265 V=150.0
MOVC C00266 EC00266 V=150.0
MOVC C00267 EC00267 V=150.0
MOVL C00268 EC00268 V=150.0
MOVC C00269 EC00269 V=150.0
MOVC C00270 EC00270 V=150.0
MOVC C00271 EC00271 V=150.0
MOVL C00272 EC00272 V=150.0
MOVC C00273 EC00273 V=150.0
MOVC C00274 EC00274 V=150.0
MOVC C00275 EC00275 V=150.0
MOVL C00276 EC00276 V=150.0
MOVC C00277 EC00277 V=150.0
MOVC C00278 EC00278 V=150.0
MOVC C00279 EC00279 V=150.0
MOVL C00280 EC00280 V=150.0
MOVC C00281 EC00281 V=150.0
MOVC C00282 EC00282 V=150.0
MOVC C00283 EC00283 V=150.0
MOVL C00284 EC00284 V=150.0
MOVC C00285 EC00285 V=150.0
MOVC C00286 EC00286 V=150.0
MOVC C00287 EC00287 V=150.0
MOVL C00288 EC00288 V=150.0
MOVC C00289 EC00289 V=150.0
MOVC C00290 EC00290 V=150.0
MOVC C00291 EC00291 V=150.0
MOVL C00292 EC00292 V=150.0
MOVC C00293 EC00293 V=150.0
MOVC C00294 EC00294 V=150.0
MOVC C00295 EC00295 V=150.0
MOVL C00296 EC00296 V=150.0
MOVC C00297 EC00297 V=150.0
MOVC C00298 EC00298 V=150.0
MOVC C00299 EC00299 V=150.0
MOVL C00300 EC00300 V=150.0
MOVC C00301 EC00301 V=150.0
MOVC C00302 EC00302 V=150.0
MOVC C00303 EC00303 V=150.0
MOVL C00304 EC00304 V=150.0
MOVC C00305 EC00305 V=150.0
MOVC C00306 EC00306 V=150.0
MOVC C00307 EC00307 V=150.0
MOVL C00308 EC00308 V=150.0
MOVC C00309 EC00309 V=150.0
MOVC C00310 EC00310 V=150.0
MOVC C00311 EC00311 V=150.0
MOVL C00312 EC00312 V=150.0
MOVC C00313 EC00313 V=150.0
MOVC C00314 EC00314 V=150.0
MOVC C00315 EC00315 V=150.0
MOVL C00316 EC00316 V=150.0
MOVC C00317 EC00317 V=150.0
MOVC C00318 EC00318 V=150.0
MOVC C00319 EC00319 V=150.0
MOVL C00320 EC00320 V=150.0
MOVC C00321 EC00321 V=150.0
MOVC C00322 EC00322 V=150.0
MOVC C00323 EC00323 V=150.0
MOVL C00324 EC00324 V=150.0
MOVC C00325 EC00325 V=150.0
MOVC C00326 EC00326 V=150.0
MOVC C00327 EC00327 V=150.0
MOVL C00328 EC00328 V=150.0
MOVC C00329 EC00329 V=150.0
MOVC C00330 EC00330 V=150.0
MOVC C00331 EC00331 V=150.0
MOVL C00332 EC00332 V=150.0
MOVC C00333 EC00333 V=150.0
MOVC C00334 EC00334 V=150.0
MOVC C00335 EC00335 V=150.0
MOVL C00336 EC00336 V=150.0
MOVC C00337 EC00337 V=150.0
MOVC C00338 EC00338 V=150.0
MOVC C00339 EC00339 V=150.0
MOVL C00340 EC00340 V=150.0
MOVC C00341 EC00341 V=150.0
MOVC C00342 EC00342 V=150.0
MOVC C00343 EC00343 V=150.0
MOVL C00344 EC00344 V=150.0
MOVC C00345 EC00345 V=150.0
MOVC C00346 EC00346 V=150.0
MOVC C00347 EC00347 V=150.0
MOVL C00348 EC00348 V=150.0
MOVC C00349 EC00349 V=150.0
MOVC C00350 EC00350 V=150.0
MOVC C00351 EC00351 V=150.0
MOVL C00352 EC00352 V=150.0
MOVC C00353 EC00353 V=150.0
MOVC C00354 EC00354 V=150.0
MOVC C00355 EC00355 V=150.0
MOVL C00356 EC00356 V=150.0
MOVC C00357 EC00357 V=150.0
MOVC C00358 EC00358 V=150.0
MOVC C00359 EC00359 V=150.0
MOVL C00360 EC00360 V=150.0
MOVC C00361 EC00361 V=150.0
MOVC C00362 EC00362 V=150.0
MOVC C00363 EC00363 V=150.0
MOVL C00364 EC00364 V=150.0
MOVC C00365 EC00365 V=150.0
MOVC C00366 EC00366 V=150.0
MOVC C00367 EC00367 V=150.0
MOVL C00368 EC00368 V=150.0
MOVC C00369 EC00369 V=150.0
MOVC C00370 EC00370 V=150.0
MOVC C00371 EC00371 V=150.0
MOVL C00372 EC00372 V=150.0
MOVC C00373 EC00373 V=150.0
MOVC C00374 EC00374 V=150.0
MOVC C00375 EC00375 V=150.0
MOVL C00376 EC00376 V=150.0
MOVC C00377 EC00377 V=150.0
MOVC C00378 EC00378 V=150.0
MOVC C00379 EC00379 V=150.0
MOVL C00380 EC00380 V=150.0
MOVC C00381 EC00381 V=150.0
MOVC C00382 EC00382 V=150.0
MOVC C00383 EC00383 V=150.0
CALL JOB:SPYOF
MOVJ P009 VJ=15.00
MOVL P009 EX002 V=150.0
MOVJ C00384 EC00384 VJ=15.00
CALL JOB:SPYON
MOVC C00385 EC00385 V=150.0
MOVC C00386 EC00386 V=150.0
MOVC C00387 EC00387 V=150.0
MOVL C00388 EC00388 V=150.0
MOVC C00389 EC00389 V=150.0
MOVC C00390 EC00390 V=150.0
MOVC C00391 EC00391 V=150.0
MOVL C00392 EC00392 V=150.0
MOVC C00393 EC00393 V=150.0
MOVC C00394 EC00394 V=150.0
MOVC C00395 EC00395 V=150.0
MOVL C00396 EC00396 V=150.0
MOVC C00397 EC00397 V=150.0
MOVC C00398 EC00398 V=150.0
MOVC C00399 EC00399 V=150.0
MOVL C00400 EC00400 V=150.0
MOVC C00401 EC00401 V=150.0
MOVC C00402 EC00402 V=150.0
MOVC C00403 EC00403 V=150.0
MOVL C00404 EC00404 V=150.0
MOVC C00405 EC00405 V=150.0
MOVC C00406 EC00406 V=150.0
MOVC C00407 EC00407 V=150.0
MOVL C00408 EC00408 V=150.0
MOVC C00409 EC00409 V=150.0
MOVC C00410 EC00410 V=150.0
MOVC C00411 EC00411 V=150.0
MOVL C00412 EC00412 V=150.0
MOVC C00413 EC00413 V=150.0
MOVC C00414 EC00414 V=150.0
MOVC C00415 EC00415 V=150.0
MOVL C00416 EC00416 V=150.0
MOVC C00417 EC00417 V=150.0
MOVC C00418 EC00418 V=150.0
MOVC C00419 EC00419 V=150.0
MOVL C00420 EC00420 V=150.0
MOVC C00421 EC00421 V=150.0
MOVC C00422 EC00422 V=150.0
MOVC C00423 EC00423 V=150.0
MOVL C00424 EC00424 V=150.0
MOVC C00425 EC00425 V=150.0
MOVC C00426 EC00426 V=150.0
MOVC C00427 EC00427 V=150.0
MOVL C00428 EC00428 V=150.0
MOVC C00429 EC00429 V=150.0
MOVC C00430 EC00430 V=150.0
MOVC C00431 EC00431 V=150.0
MOVL C00432 EC00432 V=150.0
MOVC C00433 EC00433 V=150.0
MOVC C00434 EC00434 V=150.0
MOVC C00435 EC00435 V=150.0
MOVL C00436 EC00436 V=150.0
MOVC C00437 EC00437 V=150.0
MOVC C00438 EC00438 V=150.0
MOVC C00439 EC00439 V=150.0
MOVL C00440 EC00440 V=150.0
MOVC C00441 EC00441 V=150.0
MOVC C00442 EC00442 V=150.0
MOVC C00443 EC00443 V=150.0
MOVL C00444 EC00444 V=150.0
MOVC C00445 EC00445 V=150.0
MOVC C00446 EC00446 V=150.0
MOVC C00447 EC00447 V=150.0
MOVL C00448 EC00448 V=150.0
MOVC C00449 EC00449 V=150.0
MOVC C00450 EC00450 V=150.0
MOVC C00451 EC00451 V=150.0
MOVL C00452 EC00452 V=150.0
MOVC C00453 EC00453 V=150.0
MOVC C00454 EC00454 V=150.0
MOVC C00455 EC00455 V=150.0
MOVL C00456 EC00456 V=150.0
MOVC C00457 EC00457 V=150.0
MOVC C00458 EC00458 V=150.0
MOVC C00459 EC00459 V=150.0
MOVL C00460 EC00460 V=150.0
MOVC C00461 EC00461 V=150.0
MOVC C00462 EC00462 V=150.0
MOVC C00463 EC00463 V=150.0
MOVL C00464 EC00464 V=150.0
MOVC C00465 EC00465 V=150.0
MOVC C00466 EC00466 V=150.0
MOVC C00467 EC00467 V=150.0
MOVL C00468 EC00468 V=150.0
MOVC C00469 EC00469 V=150.0
MOVC C00470 EC00470 V=150.0
MOVC C00471 EC00471 V=150.0
MOVL C00472 EC00472 V=150.0
MOVC C00473 EC00473 V=150.0
MOVC C00474 EC00474 V=150.0
MOVC C00475 EC00475 V=150.0
MOVL C00476 EC00476 V=150.0
MOVC C00477 EC00477 V=150.0
MOVC C00478 EC00478 V=150.0
MOVC C00479 EC00479 V=150.0
MOVL C00480 EC00480 V=150.0
MOVC C00481 EC00481 V=150.0
MOVC C00482 EC00482 V=150.0
MOVC C00483 EC00483 V=150.0
MOVL C00484 EC00484 V=150.0
MOVC C00485 EC00485 V=150.0
MOVC C00486 EC00486 V=150.0
MOVC C00487 EC00487 V=150.0
CALL JOB:SPYOF
MOVJ P009 VJ=15.00
MOVL P009 EX003 V=150.0
END
